TYPE ST_LinearReport :
STRUCT
	ID_Linear  : INT;
    pump1      : STRING(100);
    pump2      : STRING(100);
    pump3      : STRING(100);
    pump4      : STRING(100);
    pump5      : STRING(100);
    pump6      : STRING(100);
    pump7      : STRING(100);
    pump8      : STRING(100);
    pump9      : STRING(100);
    pump10     : STRING(100);
    changedBy  : STRING(100);
    changedOn  : STRING(100);
END_STRUCT
END_TYPE

(* stored: Version 1.1.0.1, ProductVersion 3.1.4024.15
   DUT ST_LinearReport: Id {22fa49d8-b62b-40f5-a17c-3784f31ce2ed} *)
